FUNCTION_BLOCK T_TestBase EXTENDS T_NamedBase
VAR
	_done : BOOL;
	_testsPassed : BOOL;
	_reset : BOOL;
	_startTests : BOOL;
	_task : T_Task;
	_startTime : LINT; // ms
END_VAR

{attribute 'monitoring' := 'call'} PROPERTY Done : BOOL;
GET
Done := _done;
END_GET
SET
_done := Done;
END_SET
END_PROPERTY

{attribute 'monitoring' := 'call'} PROPERTY DonePulse : BOOL
GET
VAR_INST
	pulse : R_TRIG;
END_VAR
pulse( CLK := Done );
DonePulse := pulse.Q;
END_GET
END_PROPERTY

{attribute 'monitoring' := 'call'} PROPERTY nElapsedTimeInMs : LINT
GET
nElapsedTimeInMs := _task.DistributedClockTimeInMs - _startTime;
END_GET
END_PROPERTY

{attribute 'monitoring' := 'call'} PROPERTY Passed : BOOL;
GET
Passed := THIS^._testsPassed AND Done;
END_GET
END_PROPERTY

METHOD Reset
_reset := TRUE;
END_METHOD

METHOD Start
THIS^.Reset();
_startTests := TRUE;
END_METHOD

METHOD StartTimer
_task.SetToThisTask(); // which ever thread this is called on sets the timer.
_startTime := _task.DistributedClockTimeInMs;
END_METHOD

{attribute 'monitoring' := 'call'} PROPERTY tElapsedTimeInMs : TIME
GET
tElapsedTimeInMs := TO_TIME(nElapsedTimeInMs);
END_GET
END_PROPERTY

END_FUNCTION_BLOCK

(* stored: Version 1.1.0.1, ProductVersion 3.1.4022.18
   POU T_TestBase: Id {cf43b595-fd8d-4755-bf5a-2fec59bd2fc0}, SpecialFunc None
   Property Done: Id {cc6b35ed-861e-40d9-b64a-583b9efa7f70}
   Get Get: Id {563a55d2-6394-4feb-9952-e27846a74973}
   Set Set: Id {cd6bb8e0-1035-4620-99d7-fe63791219ff}
   Property DonePulse: Id {69daae97-218a-4a5e-a596-88e585acbc2a}
   Get Get: Id {bb5d7734-e305-4edc-91b9-025e213ca3a1}
   Property nElapsedTimeInMs: Id {e45e4b5b-34f4-4a70-ba84-9331932690c9}
   Get Get: Id {f0416f8b-05b8-41ce-8c39-e6b4ca45df62}
   Property Passed: Id {bbf31e0e-e0e1-4439-bc58-ff8a8d786e36}
   Get Get: Id {c2a05465-df13-4139-940b-78df6bfb865e}
   Method Reset: Id {ed97f53b-fcfb-4b50-86ef-8defedbb18c2}
   Method Start: Id {46534931-5501-419a-b28c-8c4d057122da}
   Method StartTimer: Id {d4d9a5ca-456e-412d-b8dc-70d4c2039c9a}
   Property tElapsedTimeInMs: Id {a7b4614d-a01c-4463-8818-40a516e5640b}
   Get Get: Id {dc2255c6-8bf8-48a6-b1a6-fd6bfa69bf11} *)
